Yaskawa INFORM job: clamp_07_08_23_planes_program.JBI

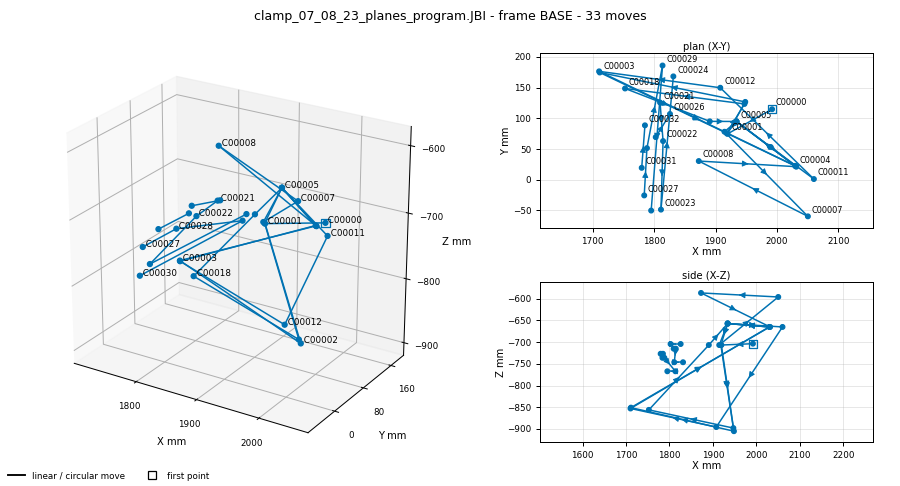
[picture p0: tool path of clamp_07_08_23_planes_program.JBI in frame BASE, 33 of 39 moves have a stored position in this frame; points joined in program order, loops and branches not executed]
/JOB
//NAME clamp_07_08_23_planes_program
//POS
///NPOS 33,0,33,0,0,0
///TOOL 0
///POSTYPE BASE
///RECTAN
///RCONF 0,0,0,0,0,0,0,0,0,0,0,0,0,0,0,0,0,0,0,0,0,0,0,0
C00000=1992.090525,114.888600,-703.733050,175.000000,-60.100974,-93.452339
C00001=1919.472395,74.766857,-706.834963,-175.000000,-61.458604,-51.021412
C00002=1948.389959,126.804095,-905.101865,180.000000,-60.000000,0.000000
C00003=1711.399645,174.688909,-850.854389,180.000000,-60.000000,0.000000
C00004=2030.633745,21.975728,-665.209748,175.000000,-40.948846,-175.000000
C00005=1934.016934,94.892200,-657.368686,175.000000,-36.140931,-78.595303
C00006=1914.580766,78.214768,-706.834963,175.000000,-61.458604,-51.021412
C00007=2050.383094,-59.601278,-596.243401,-175.000000,20.870044,5.000000
C00008=1872.707848,30.456483,-586.952789,159.479170,-22.066643,8.004362
C00009=2031.587247,21.303643,-665.209748,175.000000,-40.948846,-175.000000
C00010=1934.016934,94.892200,-657.368686,175.000000,-36.140931,-78.595303
C00011=2060.160095,1.163799,-665.209748,175.000000,-40.948846,-175.000000
C00012=1907.728501,149.857467,-895.542268,180.000000,-60.000000,0.000000
C00013=1710.387298,176.564685,-852.833905,180.000000,-60.000000,0.000000
C00014=2029.588790,22.712275,-665.209748,-175.000000,-40.948846,-175.000000
C00015=1934.016934,94.892200,-657.368686,175.000000,-36.140931,-78.595303
C00016=1918.285397,75.603524,-706.834963,175.000000,-61.458604,-51.021412
C00017=1947.086668,123.492292,-897.887528,180.000000,-60.000000,0.000000
C00018=1752.627980,148.657220,-856.021720,180.000000,-60.000000,0.000000
C00019=1890.584918,95.128471,-706.834963,175.000000,-61.458604,-51.021412
C00020=1934.016934,94.892200,-657.368686,175.000000,-36.140931,-78.595303
C00021=1809.644350,125.753900,-715.113810,180.000000,-60.000000,0.000000
C00022=1814.544350,62.998300,-715.113810,180.000000,-60.000000,0.000000
C00023=1811.124350,-48.630600,-746.419310,180.000000,-60.000000,0.000000
C00024=1831.304350,168.344900,-746.419310,180.000000,-60.000000,0.000000
C00025=1802.593540,69.430140,-704.453900,175.000000,-59.609272,-5.000000
C00026=1825.811400,107.130140,-704.453900,175.000000,-59.609272,-5.000000
C00027=1783.852150,-25.534339,-736.105660,180.000000,-60.000000,0.000000
C00028=1788.272150,51.492662,-736.105660,180.000000,-60.000000,0.000000
C00029=1813.662150,186.043161,-767.225160,180.000000,-60.000000,0.000000
C00030=1795.162150,-50.185439,-767.225160,180.000000,-60.000000,0.000000
C00031=1779.746900,19.425775,-726.886720,180.000000,-60.000000,0.000000
C00032=1785.015300,88.655775,-726.886720,180.000000,-60.000000,0.000000
///POSTYPE PULSE
///PULSE
EC00000=0
EC00001=0
EC00002=0
EC00003=0
EC00004=0
EC00005=0
EC00006=0
EC00007=0
EC00008=0
EC00009=0
EC00010=0
EC00011=0
EC00012=0
EC00013=0
EC00014=0
EC00015=0
EC00016=0
EC00017=0
EC00018=0
EC00019=0
EC00020=0
EC00021=0
EC00022=0
EC00023=0
EC00024=0
EC00025=92160
EC00026=92160
EC00027=184320
EC00028=184320
EC00029=184320
EC00030=184320
EC00031=276480
EC00032=276480
//INST
///DATE 2023/08/07 12:02
///ATTR SC,RW,RJ
////FRAME BASE
///GROUP1 RB1,ST1
NOP
MOVJ P009 EX000 VJ=15.00
MOVJ C00000 EC00000 VJ=15.0
CALL JOB:SPYON
MOVL C00001 EC00001 V=150.0
MOVL C00002 EC00002 V=150.0
MOVL C00003 EC00003 V=150.0
MOVL C00004 EC00004 V=150.0
MOVL C00005 EC00005 V=150.0
MOVL C00006 EC00006 V=150.0
MOVL C00007 EC00007 V=150.0
MOVL C00008 EC00008 V=150.0
MOVL C00009 EC00009 V=150.0
MOVL C00010 EC00010 V=150.0
MOVL C00011 EC00011 V=150.0
MOVL C00012 EC00012 V=150.0
MOVL C00013 EC00013 V=150.0
MOVL C00014 EC00014 V=150.0
MOVL C00015 EC00015 V=150.0
MOVL C00016 EC00016 V=150.0
MOVL C00017 EC00017 V=150.0
MOVL C00018 EC00018 V=150.0
MOVL C00019 EC00019 V=150.0
MOVL C00020 EC00020 V=150.0
CALL JOB:SPYOF
MOVJ P009 VJ=15.00
MOVJ C00021 EC00021 VJ=15.0
CALL JOB:SPYON
MOVL C00022 EC00022 V=150.0
MOVL C00023 EC00023 V=150.0
MOVL C00024 EC00024 V=150.0
CALL JOB:SPYOF
MOVJ P009 VJ=15.00
MOVJ C00025 EC00025 VJ=15.0
CALL JOB:SPYON
MOVL C00026 EC00026 V=150.0
CALL JOB:SPYOF
MOVJ P009 VJ=15.00
MOVJ C00027 EC00027 VJ=15.0
CALL JOB:SPYON
MOVL C00028 EC00028 V=150.0
MOVL C00029 EC00029 V=150.0
MOVL C00030 EC00030 V=150.0
CALL JOB:SPYOF
MOVJ P009 VJ=15.00
MOVJ C00031 EC00031 VJ=15.0
CALL JOB:SPYON
MOVL C00032 EC00032 V=150.0
CALL JOB:SPYOF
MOVJ P009 VJ=15.00
END
